FUNCTION_BLOCK TestADSLogger EXTENDS TcUnit.FB_TestSuite
VAR_INPUT
END_VAR
VAR_OUTPUT
END_VAR
VAR
END_VAR

submit_info();
submit_warning();
submit_error();
submit_alarm();
change_default_level_to_warning_and_submit_info();
change_default_level_to_warning_and_submit_error();
create_event_with_a_parameter();
create_runner_message_with_a_parameter();

METHOD change_default_level_to_warning_and_submit_error
VAR_INPUT
END_VAR
VAR_INST
  sut: ADSLoggerTestsystem;
END_VAR
TEST('Change default level to warning and submit error');

sut.runner.add_logger(sut.logger);
sut.logger.level := EventLevel.WARNING;
sut.event.message := 'Default level warning';
sut.event.error();

AssertEquals_DWORD(ADSLOG_MSGTYPE_ERROR, sut.logger.mask, '');
AssertEquals_STRING(' | Error: ', sut.logger.prefix, '');
AssertEquals_STRING(' | Error: Default level warning', sut.logger.formatted_output, '');

TEST_FINISHED();
END_METHOD

METHOD change_default_level_to_warning_and_submit_info
VAR_INPUT
END_VAR
VAR_INST
  sut: ADSLoggerTestsystem;
END_VAR
TEST('Change default level to warning and submit info');

sut.runner.add_logger(sut.logger);
sut.logger.level := EventLevel.WARNING;
sut.event.message := 'Default level warning';
sut.event.info();

AssertEquals_DWORD(0, sut.logger.mask, '');
AssertEquals_STRING('', sut.logger.prefix, '');
AssertEquals_STRING('', sut.logger.formatted_output, '');

TEST_FINISHED();
END_METHOD

METHOD create_event_with_a_parameter
VAR_INST
  sut: ADSLoggerTestsystem;
END_VAR
VAR
  parameter: INT;
END_VAR
TEST('Create event with a parameter');

sut.runner.add_logger(sut.logger);
sut.event.message := 'Test %d';
parameter := 123;
sut.event.parameter := F_INT(parameter);
sut.event.error();

AssertEquals_DWORD(ADSLOG_MSGTYPE_ERROR, sut.logger.mask, '');
AssertEquals_STRING(' | Error: ', sut.logger.prefix, '');
AssertEquals_STRING(' | Error: Test 123', sut.logger.formatted_output, '');

TEST_FINISHED();
END_METHOD

METHOD create_runner_message_with_a_parameter
VAR_INST
  sut: ADSLoggerTestsystem;
END_VAR
VAR
  parameter: REAL;
END_VAR
TEST('Create runner message with a parameter');

sut.runner.add_logger(sut.logger);
parameter := 3.14;
sut.runner.parameter := F_REAL(parameter);
sut.runner.warning(message:='Test %1.2f');

AssertEquals_STRING(' | Warning: Test 3.14', sut.logger.formatted_output, '');

TEST_FINISHED();
END_METHOD

METHOD submit_alarm
VAR_INPUT
END_VAR
VAR_INST
  sut: ADSLoggerTestsystem;
END_VAR
TEST('Submit alarm');

sut.runner.add_logger(sut.logger);
sut.event.message := 'Alarm';
sut.event.alarm();

AssertEquals_DWORD(ADSLOG_MSGTYPE_ERROR, sut.logger.mask, '');
AssertEquals_STRING(' | Error: ', sut.logger.prefix, '');
AssertEquals_STRING(' | Error: Alarm', sut.logger.formatted_output, '');

TEST_FINISHED();
END_METHOD

METHOD submit_error
VAR_INPUT
END_VAR
VAR_INST
  sut: ADSLoggerTestsystem;
END_VAR
TEST('Submit error');

sut.runner.add_logger(sut.logger);
sut.event.message := 'Error';
sut.event.error();

AssertEquals_DWORD(ADSLOG_MSGTYPE_ERROR, sut.logger.mask, '');
AssertEquals_STRING(' | Error: ', sut.logger.prefix, '');
AssertEquals_STRING(' | Error: Error', sut.logger.formatted_output, '');

TEST_FINISHED();
END_METHOD

METHOD submit_info
VAR_INPUT
END_VAR
VAR_INST
  sut: ADSLoggerTestsystem;
END_VAR
TEST('Submit info');

sut.runner.add_logger(sut.logger);
sut.event.message := 'Info';
sut.event.info();

AssertEquals_DWORD(ADSLOG_MSGTYPE_HINT, sut.logger.mask, '');
AssertEquals_STRING(' | Info: ', sut.logger.prefix, '');
AssertEquals_STRING(' | Info: Info', sut.logger.formatted_output, '');

TEST_FINISHED();
END_METHOD

METHOD submit_warning
VAR_INPUT
END_VAR
VAR_INST
  sut: ADSLoggerTestsystem;
END_VAR
TEST('Submit warning');

sut.runner.add_logger(sut.logger);
sut.event.message := 'Warning';
sut.event.warning();

AssertEquals_DWORD(ADSLOG_MSGTYPE_WARN, sut.logger.mask, '');
AssertEquals_STRING(' | Warning: ', sut.logger.prefix, '');
AssertEquals_STRING(' | Warning: Warning', sut.logger.formatted_output, '');

TEST_FINISHED();
END_METHOD

END_FUNCTION_BLOCK

(* stored: Version 1.1.0.1, ProductVersion 3.1.4024.9
   POU TestADSLogger: Id {e126a8bd-dc53-47fb-b987-2c50fb609a8b}, SpecialFunc None
   Method change_default_level_to_warning_and_submit_error: Id {fde893c3-5a5b-4fdb-ab58-28f4712e9db3}
   Method change_default_level_to_warning_and_submit_info: Id {559af52a-7fea-4e0d-91b3-752a3aa7dcc3}
   Method create_event_with_a_parameter: Id {220a2117-cff1-4bcc-9fe0-a73e4a8b7629}
   Method create_runner_message_with_a_parameter: Id {e52eac1d-cb65-49b4-bc09-5d81f556beb4}
   Method submit_alarm: Id {7203e8ee-f5fe-4e56-af12-ce30cf3bab16}
   Method submit_error: Id {7c89dd55-cac3-43cf-b229-89629492e809}
   Method submit_info: Id {bd81e84a-3e0d-47ff-97fa-d790029e78ab}
   Method submit_warning: Id {d791f11d-b6d0-4afa-8f91-e5b068e59d16} *)
